FUNCTION TryConvert_REAL_TO_LINT : BOOL
VAR_INPUT
	in : REAL;
	out : REFERENCE TO LINT;
END_VAR

IF in > DatatypeLimits.MAX_VALUE_OF_REAL_WHICH_CAN_BE_HELD_IN_A_LINT THEN
	RETURN;
END_IF

IF in < DatatypeLimits.MIN_VALUE_OF_REAL_WHICH_CAN_BE_HELD_IN_A_LINT THEN
	RETURN;
END_IF

out := REAL_TO_LINT(in);
TryConvert_REAL_TO_LINT := TRUE;

END_FUNCTION

(* stored: Version 1.1.0.1, ProductVersion 3.1.4024.12
   POU TryConvert_REAL_TO_LINT: Id {f670c016-3b24-4717-8583-0300217dedba}, SpecialFunc None *)
